SUBAPPLICATION Uebung_003a0 (* DigitalInput_I1/_I2 auf DigitalOutput_Q1/_I2 - mit untyped Subapp *)
  (* Standard: 61499-2; Description: Copyright (c) 2023 Meisterschulen am Ostbahnhof This program and the accompanying materials are made available under the terms of the Eclipse Public License 2.0 which is available at https://www.eclipse.org/legal/epl-2.0/ SPDX-License-Identifier: EPL-2.0 *)
  (* Version 1.0, 2023-10-23, Franz Höpfinger, Meisterschulen am Ostbahnhof, initial API and implementation and/or initial documentation *)
  PACKAGE Uebungen;
  IMPORT logiBUS::io::DI::logiBUS_DI::Input_I1;
  IMPORT logiBUS::io::DI::logiBUS_DI::Input_I2;
  IMPORT logiBUS::io::DQ::logiBUS_DO::Output_Q1;
  IMPORT logiBUS::io::DQ::logiBUS_DO::Output_Q2;
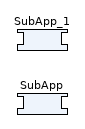
  SUBAPPLICATION SubApp
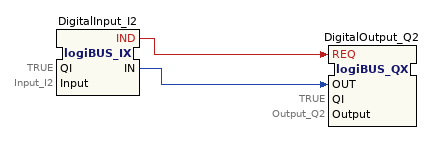
    FBS
      DigitalInput_I2 : logiBUS::io::DI::logiBUS_IX(QI := TRUE, Input := Input_I2);
      DigitalOutput_Q2 : logiBUS::io::DQ::logiBUS_QX(QI := TRUE, Output := Output_Q2);
    END_FBS
    EVENT_CONNECTIONS
      DigitalInput_I2.IND TO DigitalOutput_Q2.REQ;
    END_CONNECTIONS
    DATA_CONNECTIONS
      DigitalInput_I2.IN TO DigitalOutput_Q2.OUT;
    END_CONNECTIONS
  END_SUBAPPLICATION
  SUBAPPLICATION SubApp_1
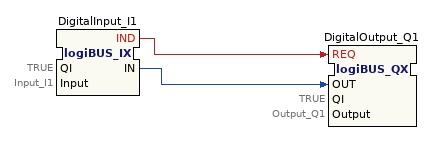
    FBS
      DigitalOutput_Q1 : logiBUS::io::DQ::logiBUS_QX(QI := TRUE, Output := Output_Q1);
      DigitalInput_I1 : logiBUS::io::DI::logiBUS_IX(QI := TRUE, Input := Input_I1);
    END_FBS
    EVENT_CONNECTIONS
      DigitalInput_I1.IND TO DigitalOutput_Q1.REQ;
    END_CONNECTIONS
    DATA_CONNECTIONS
      DigitalInput_I1.IN TO DigitalOutput_Q1.OUT;
    END_CONNECTIONS
  END_SUBAPPLICATION
END_SUBAPPLICATION
